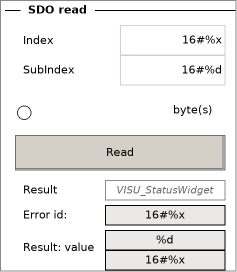
VISUALIZATION VISU_FaulhaberDrive_SDORead  // 237x272
VAR_IN_OUT
	drive : FaulhaberDrive;
    widget : FaulhaberDriveWidget;
END_VAR
    Label (20,26 100x29), "Index"
    Button (15,135 210x35), "Read", input disabled if: drive.processes.read.statuses.enabledStatus.disabled
        OnMouseClick: execute { drive.processes.read.set.noOfBytes := widget.readNoOfBytes; drive.processes.read.do_request := TRUE; }
    Textfield (120,55 105x30), "16#%d", text variable: drive.processes.read.set.subindex, input disabled if: drive.processes.read.statuses.enabledStatus.disabled
        OnMouseClick: write the text variable via Default
    Label (20,55 100x30), "SubIndex"
    Line (5,10) (20,10)
    Label (25,0 150x20), "SDO read"
    Line (95,10) (235,10)
    Textfield (120,25 105x30), "16#%x", text variable: drive.processes.read.set.index, input disabled if: drive.processes.read.statuses.enabledStatus.disabled
        OnMouseClick: write the text variable via Default
    Frame (105,180 120x20)
        shows VISU_StatusWidget(widget := widget.sdoReadStatus)
    RadioButton (15,95 155x35), variable: widget.readNoOfBytesRadioButtonItem, input disabled if: drive.processes.read.statuses.enabledStatus.disabled
        Areas[0]: Text=1
        Areas[1]: Text=2
        Areas[2]: Text=4
    Label (170,95 55x30), "byte(s)"
    Label (20,175 80x30), "Result"
    Label (20,225 80x45), "Result: value"
    Rectangle (105,230 120x20), "%d", text variable: widget.readResultValue
    Rectangle (105,205 120x20), "16#%x", text variable: drive.processes.read.errorId
    Label (20,200 80x30), "Error id:"
    Rectangle (105,250 120x20), "16#%x", text variable: widget.readResultValue
END_VISUALIZATION

(* stored: Version 1.1.0.1, ProductVersion 3.1.4019.2
   Visu VISU_FaulhaberDrive_SDORead: Id {cf062ded-cd4b-4536-920a-ef97d95526b0} *)
